(* Logix 5000 project; controller cal1632 1756-L62 rev 16.20; software revision 16.05; part 22 of 57 *)
(* tags used below, declared in another part *)
   aaa_prs : REAL;
   FAULT : BOOL;
   p01_param_fan_zero_speed : REAL;
   p01_param_open_oven_recirc_sp : REAL;
   p01_recipe_active : recipe;
   p01_sys_scp : SYS_SCP;
   p01r09_open_oven : BOOL;
   p01r09_pb_global_reset : BOOL;
   p02_dint_from_hmi : hmi_dint;
   p11r02_shutdown_temp : BOOL;
   p11r30 : routine;
   p12r02_shutdown_temp : BOOL;
   p12r30 : routine;
   p13_ai_recirc_rpm : REAL;
   p13_ao_recirc_selected_speed : REAL;
   p13_di_recirc : acs800_di_normal;
   p13_di_recirc_fan_mtr_ts : BOOL;
   p13_di_recirc_flow_ok : BOOL;
   p13_dint_to_hmi : DINT[16];
   p13_do_recirc : acs800_do_normal;
   p13r02_shutdown_temp : BOOL;
   p13r20_state : DINT;
   p13r32 : routine;
   p13r32_pb_start : BOOL;
   p13r32_pb_stop : BOOL;
   p13r32_request_auto_run : BOOL;
   p13r32_run_permissive : BOOL;
   p13r32_timer_fault : TIMER[5];
   p13r32_timer_warning : TIMER[5];
   p13r32_vfd_stopped : BOOL;
   p19_ai_prs : REAL;
   p19_ai_tc01 : REAL;
   p19_ao_cv : REAL;
   p19_di_pump : BOOL;
   p19_di_tc01_bo : BOOL;
   p19_di_tc02_bo : BOOL;
   p19_dint_to_hmi : DINT[16];
   p19_do_pump : BOOL;
   p19_flow_input_max : REAL;
   p19_flow_input_min : REAL;
   p19_flow_output_max : REAL;
   p19_flow_output_min : REAL;
   p19_param_prs_offset : REAL;
   p19_param_tc01z : REAL;
   p19_prs_input_max : REAL;
   p19_prs_input_min : REAL;
   p19_prs_output_max : REAL;
   p19_prs_output_min : REAL;
   p19r01 : routine;
   p19r02 : routine;
   p19r02_fault_exists : BOOL;
   p19r02_timer_fault : TIMER[4];
   p19r02_timer_warning : TIMER[4];
   p19r02_unack_fault : BOOL;
   p19r02_unack_warning : BOOL;
   p19r02_warning_exists : BOOL;
   p19r03 : routine;
   p19r03_flow_scp : SYS_SCP;
   p19r03_prs_input_max : REAL;
   p19r03_prs_input_min : REAL;
   p19r03_prs_output_max : REAL;
   p19r03_prs_output_min : REAL;
   p19r03_prs_scp : SYS_SCP;
   p19r03_timer_fault : TIMER[4];
   p19r03_timer_warning : TIMER[4];
   p19r04 : routine;
   p19r04_timer_fault : TIMER[4];
   p19r04_timer_warning : TIMER[4];
   p19r05 : routine;
   p19r06 : routine;
   p19r07 : routine;
   p19r08 : routine;
   p19r09 : routine;
   p19r10 : routine;
   p19r30 : routine;
   p19r31 : routine;
   p23r02 : routine;
(* P13_Zone_3, continued *)

ROUTINE R32_Recirc_VFD   (* ladder *)
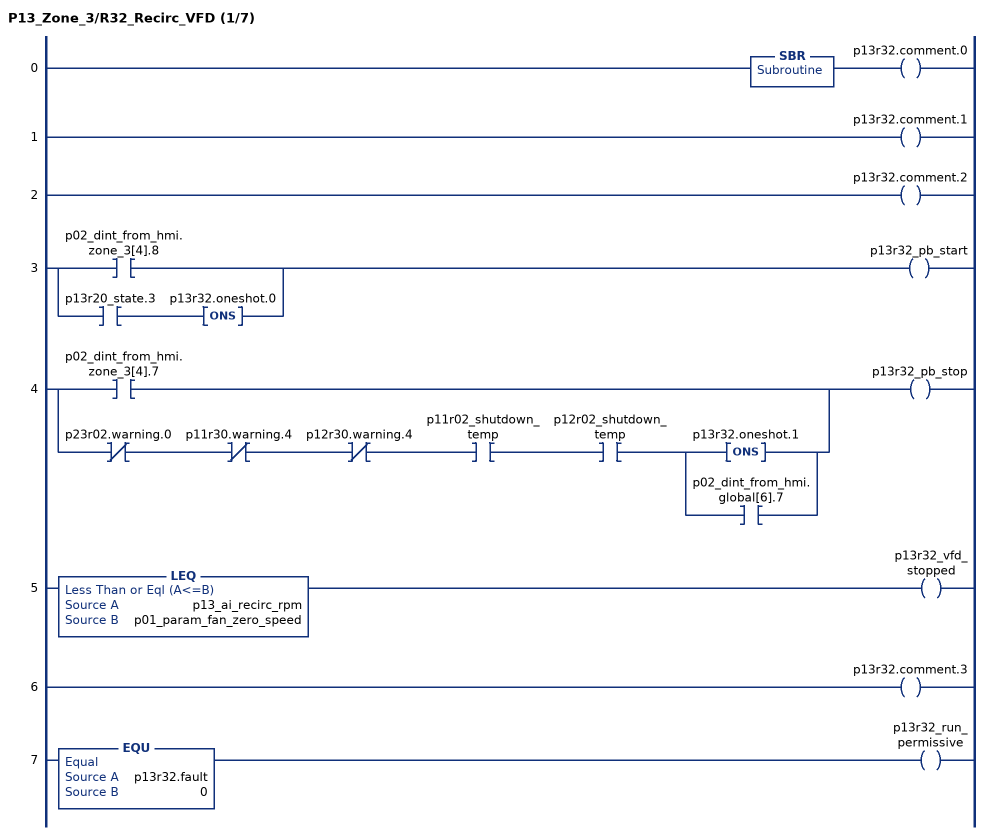
   0: SBR()OTE(p13r32.comment.0);
   1: OTE(p13r32.comment.1);
   2: OTE(p13r32.comment.2);
   3: [XIC(p02_dint_from_hmi.zone_3[4].8) ,XIC(p13r20_state.3) ONS(p13r32.oneshot.0) ]OTE(p13r32_pb_start);
   4: [XIC(p02_dint_from_hmi.zone_3[4].7) ,XIO(p23r02.warning.0) XIO(p11r30.warning.4) XIO(p12r30.warning.4) XIC(p11r02_shutdown_temp) XIC(p12r02_shutdown_temp) [ONS(p13r32.oneshot.1) ,XIC(p02_dint_from_hmi.global[6].7) ] ]OTE(p13r32_pb_stop);
   5: LEQ(p13_ai_recirc_rpm,p01_param_fan_zero_speed)OTE(p13r32_vfd_stopped);
   6: OTE(p13r32.comment.3);
   7: EQU(p13r32.fault,0)OTE(p13r32_run_permissive);
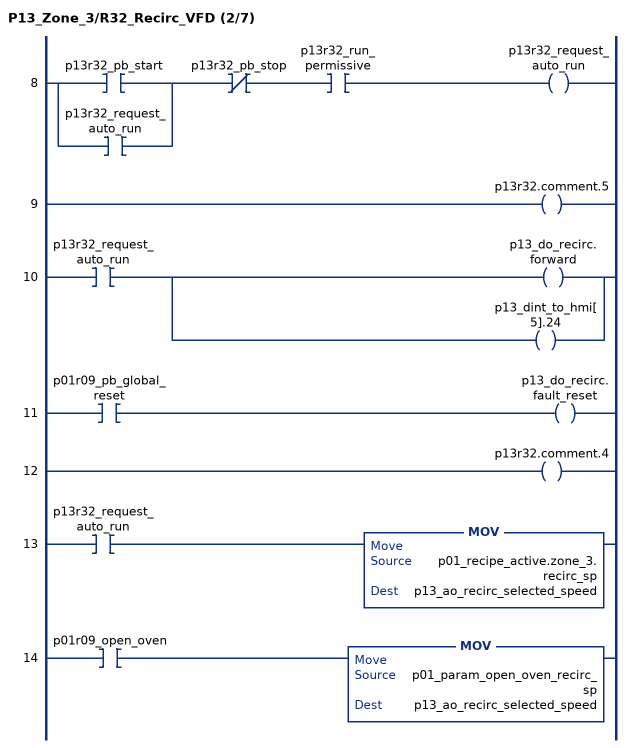
   8: [XIC(p13r32_pb_start) ,XIC(p13r32_request_auto_run) ]XIO(p13r32_pb_stop)XIC(p13r32_run_permissive)OTE(p13r32_request_auto_run);
   9: OTE(p13r32.comment.5);
   10: XIC(p13r32_request_auto_run)[OTE(p13_do_recirc.forward) ,OTE(p13_dint_to_hmi[5].24) ];
   11: XIC(p01r09_pb_global_reset)OTE(p13_do_recirc.fault_reset);
   12: OTE(p13r32.comment.4);
   13: XIC(p13r32_request_auto_run)MOV(p01_recipe_active.zone_3.recirc_sp,p13_ao_recirc_selected_speed);
   14: XIC(p01r09_open_oven)MOV(p01_param_open_oven_recirc_sp,p13_ao_recirc_selected_speed);
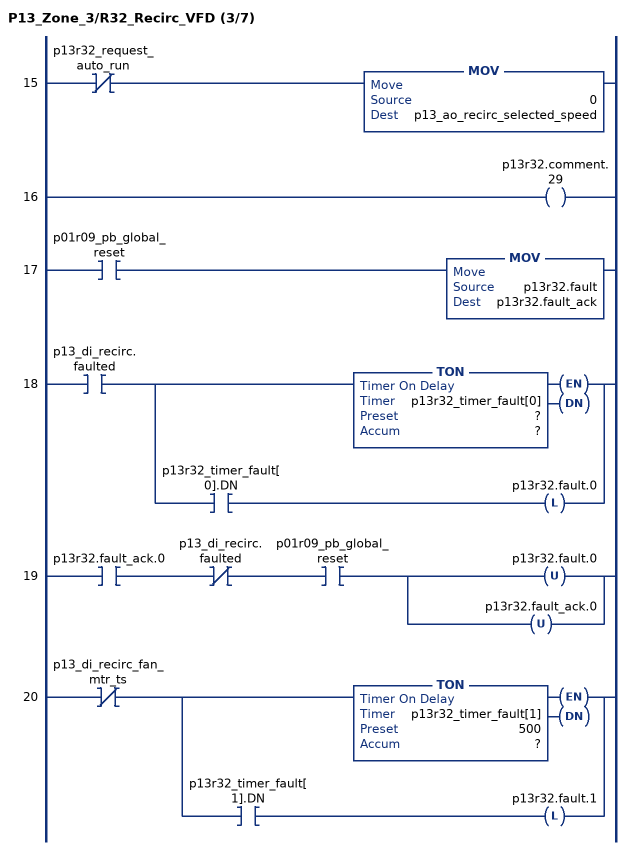
   15: XIO(p13r32_request_auto_run)MOV(0,p13_ao_recirc_selected_speed);
   16: OTE(p13r32.comment.29);
   17: XIC(p01r09_pb_global_reset)MOV(p13r32.fault,p13r32.fault_ack);
   18: XIC(p13_di_recirc.faulted)[TON(p13r32_timer_fault[0],?,?) ,XIC(p13r32_timer_fault[0].DN) OTL(p13r32.fault.0) ];
   19: XIC(p13r32.fault_ack.0)XIO(p13_di_recirc.faulted)XIC(p01r09_pb_global_reset)[OTU(p13r32.fault.0) ,OTU(p13r32.fault_ack.0) ];
   20: XIO(p13_di_recirc_fan_mtr_ts)[TON(p13r32_timer_fault[1],?,?) ,XIC(p13r32_timer_fault[1].DN) OTL(p13r32.fault.1) ];
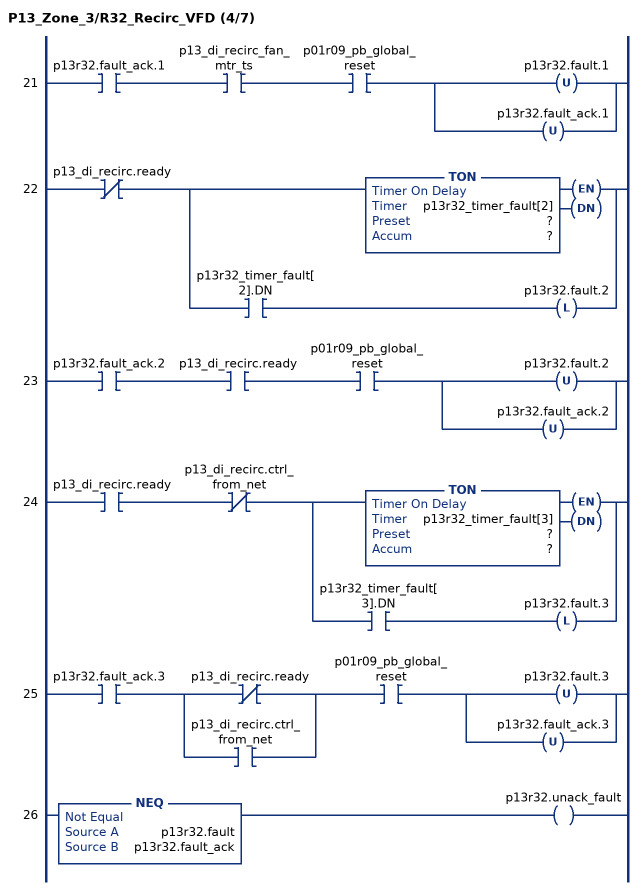
   21: XIC(p13r32.fault_ack.1)XIC(p13_di_recirc_fan_mtr_ts)XIC(p01r09_pb_global_reset)[OTU(p13r32.fault.1) ,OTU(p13r32.fault_ack.1) ];
   22: XIO(p13_di_recirc.ready)[TON(p13r32_timer_fault[2],?,?) ,XIC(p13r32_timer_fault[2].DN) OTL(p13r32.fault.2) ];
   23: XIC(p13r32.fault_ack.2)XIC(p13_di_recirc.ready)XIC(p01r09_pb_global_reset)[OTU(p13r32.fault.2) ,OTU(p13r32.fault_ack.2) ];
   24: XIC(p13_di_recirc.ready)XIO(p13_di_recirc.ctrl_from_net)[TON(p13r32_timer_fault[3],?,?) ,XIC(p13r32_timer_fault[3].DN) OTL(p13r32.fault.3) ];
   25: XIC(p13r32.fault_ack.3)[XIO(p13_di_recirc.ready) ,XIC(p13_di_recirc.ctrl_from_net) ]XIC(p01r09_pb_global_reset)[OTU(p13r32.fault.3) ,OTU(p13r32.fault_ack.3) ];
   26: NEQ(p13r32.fault,p13r32.fault_ack)OTE(p13r32.unack_fault);
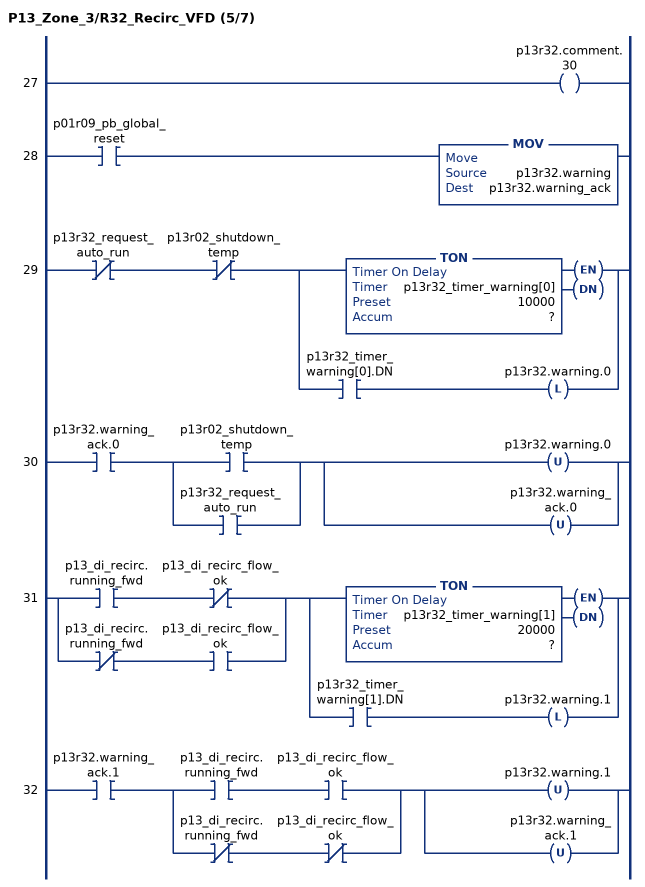
   27: OTE(p13r32.comment.30);
   28: XIC(p01r09_pb_global_reset)MOV(p13r32.warning,p13r32.warning_ack);
   29: XIO(p13r32_request_auto_run)XIO(p13r02_shutdown_temp)[TON(p13r32_timer_warning[0],?,?) ,XIC(p13r32_timer_warning[0].DN) OTL(p13r32.warning.0) ];
   30: XIC(p13r32.warning_ack.0)[XIC(p13r02_shutdown_temp) ,XIC(p13r32_request_auto_run) ][OTU(p13r32.warning.0) ,OTU(p13r32.warning_ack.0) ];
   31: [XIC(p13_di_recirc.running_fwd) XIO(p13_di_recirc_flow_ok) ,XIO(p13_di_recirc.running_fwd) XIC(p13_di_recirc_flow_ok) ][TON(p13r32_timer_warning[1],?,?) ,XIC(p13r32_timer_warning[1].DN) OTL(p13r32.warning.1) ];
   32: XIC(p13r32.warning_ack.1)[XIC(p13_di_recirc.running_fwd) XIC(p13_di_recirc_flow_ok) ,XIO(p13_di_recirc.running_fwd) XIO(p13_di_recirc_flow_ok) ][OTU(p13r32.warning.1) ,OTU(p13r32.warning_ack.1) ];
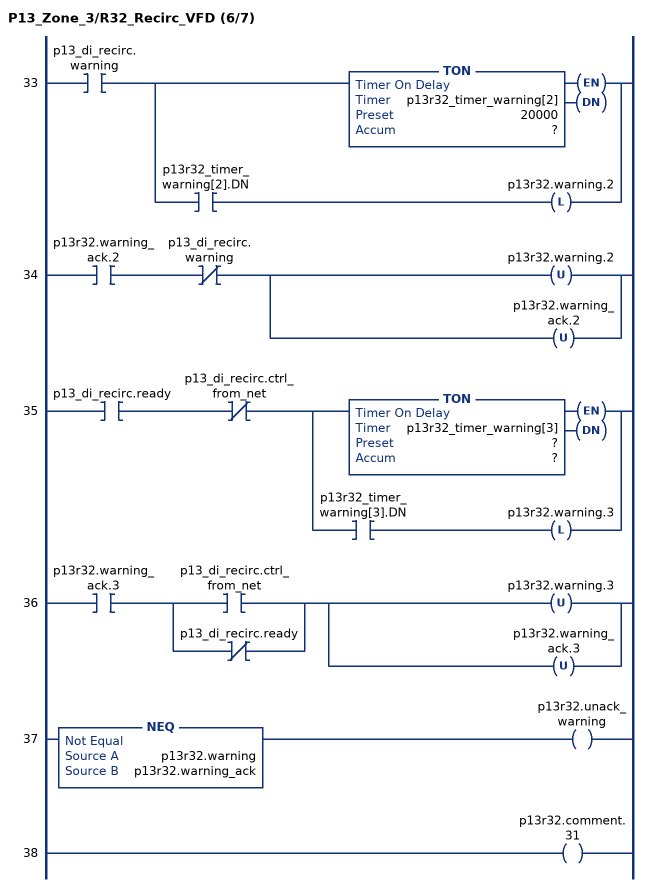
   33: XIC(p13_di_recirc.warning)[TON(p13r32_timer_warning[2],?,?) ,XIC(p13r32_timer_warning[2].DN) OTL(p13r32.warning.2) ];
   34: XIC(p13r32.warning_ack.2)XIO(p13_di_recirc.warning)[OTU(p13r32.warning.2) ,OTU(p13r32.warning_ack.2) ];
   35: XIC(p13_di_recirc.ready)XIO(p13_di_recirc.ctrl_from_net)[TON(p13r32_timer_warning[3],?,?) ,XIC(p13r32_timer_warning[3].DN) OTL(p13r32.warning.3) ];
   36: XIC(p13r32.warning_ack.3)[XIC(p13_di_recirc.ctrl_from_net) ,XIO(p13_di_recirc.ready) ][OTU(p13r32.warning.3) ,OTU(p13r32.warning_ack.3) ];
   37: NEQ(p13r32.warning,p13r32.warning_ack)OTE(p13r32.unack_warning);
   38: OTE(p13r32.comment.31);
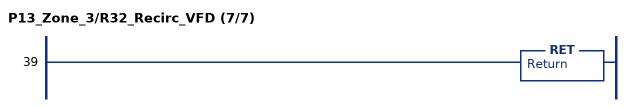
   39: RET();
END_ROUTINE
END_PROGRAM

PROGRAM P19_Advanced_Cooling   (* main routine R01_Main *)

ROUTINE R01_Main   (* ladder *)
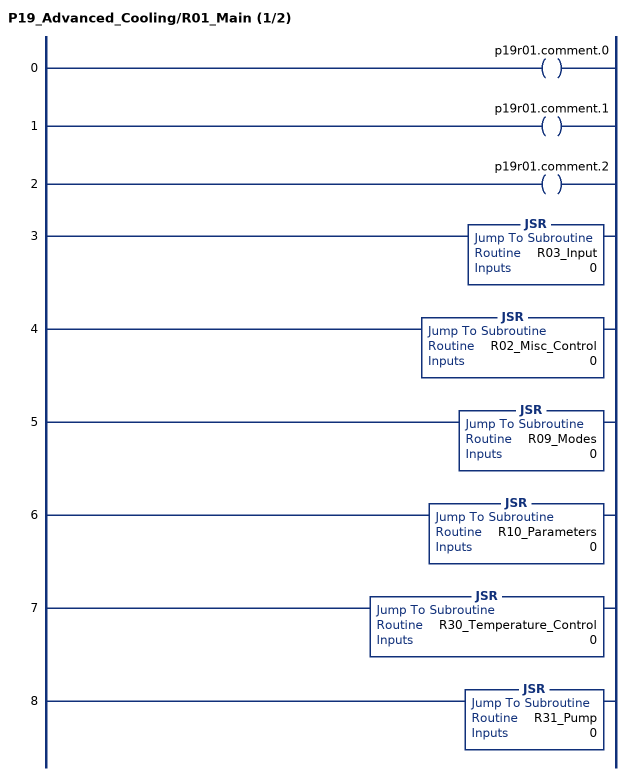
   0: OTE(p19r01.comment.0);
   1: OTE(p19r01.comment.1);
   2: OTE(p19r01.comment.2);
   3: JSR(R03_Input,0);
   4: JSR(R02_Misc_Control,0);
   5: JSR(R09_Modes,0);
   6: JSR(R10_Parameters,0);
   7: JSR(R30_Temperature_Control,0);
   8: JSR(R31_Pump,0);
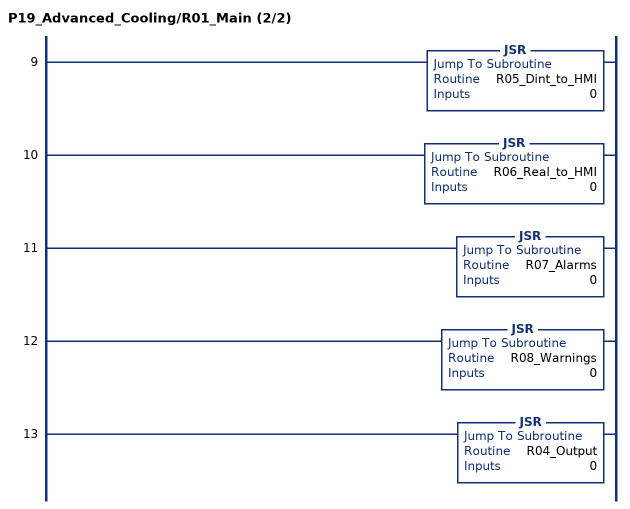
   9: JSR(R05_Dint_to_HMI,0);
   10: JSR(R06_Real_to_HMI,0);
   11: JSR(R07_Alarms,0);
   12: JSR(R08_Warnings,0);
   13: JSR(R04_Output,0);
END_ROUTINE

ROUTINE R02_Misc_Control   (* ladder *)
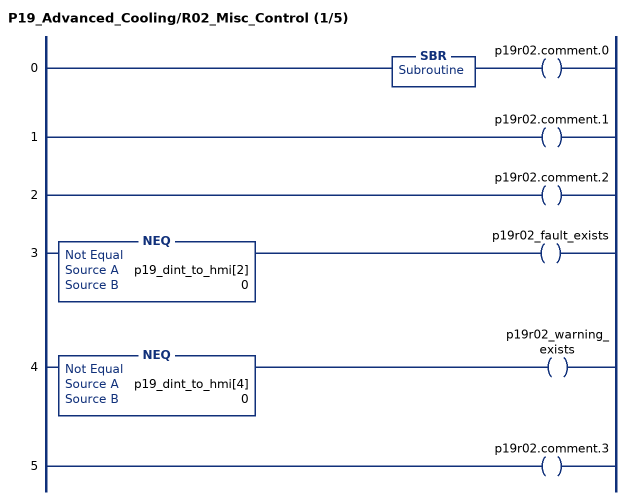
   0: SBR()OTE(p19r02.comment.0);
   1: OTE(p19r02.comment.1);
   2: OTE(p19r02.comment.2);
   3: NEQ(p19_dint_to_hmi[2],0)OTE(p19r02_fault_exists);
   4: NEQ(p19_dint_to_hmi[4],0)OTE(p19r02_warning_exists);
   5: OTE(p19r02.comment.3);
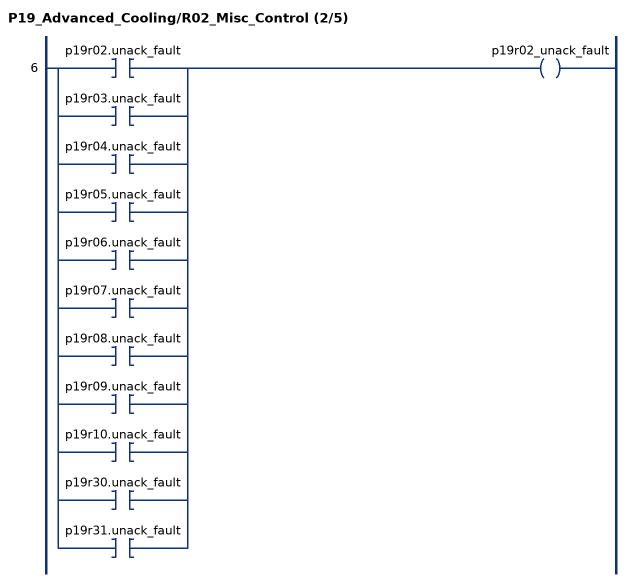
   6: [XIC(p19r02.unack_fault) ,XIC(p19r03.unack_fault) ,XIC(p19r04.unack_fault) ,XIC(p19r05.unack_fault) ,XIC(p19r06.unack_fault) ,XIC(p19r07.unack_fault) ,XIC(p19r08.unack_fault) ,XIC(p19r09.unack_fault) ,XIC(p19r10.unack_fault) ,XIC(p19r30.unack_fault) ,XIC(p19r31.unack_fault) ]OTE(p19r02_unack_fault);
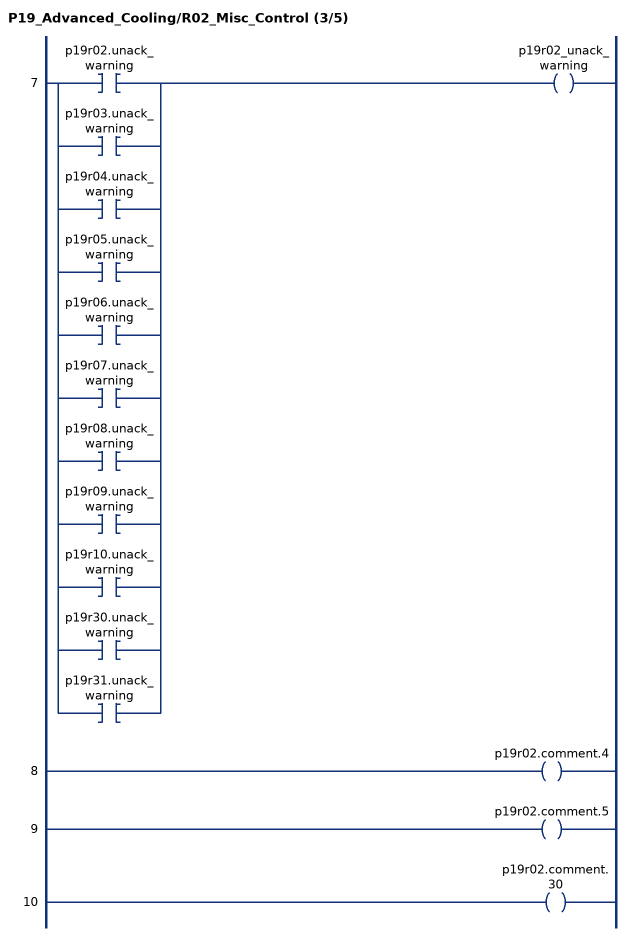
   7: [XIC(p19r02.unack_warning) ,XIC(p19r03.unack_warning) ,XIC(p19r04.unack_warning) ,XIC(p19r05.unack_warning) ,XIC(p19r06.unack_warning) ,XIC(p19r07.unack_warning) ,XIC(p19r08.unack_warning) ,XIC(p19r09.unack_warning) ,XIC(p19r10.unack_warning) ,XIC(p19r30.unack_warning) ,XIC(p19r31.unack_warning) ]OTE(p19r02_unack_warning);
   8: OTE(p19r02.comment.4);
   9: OTE(p19r02.comment.5);
   10: OTE(p19r02.comment.30);
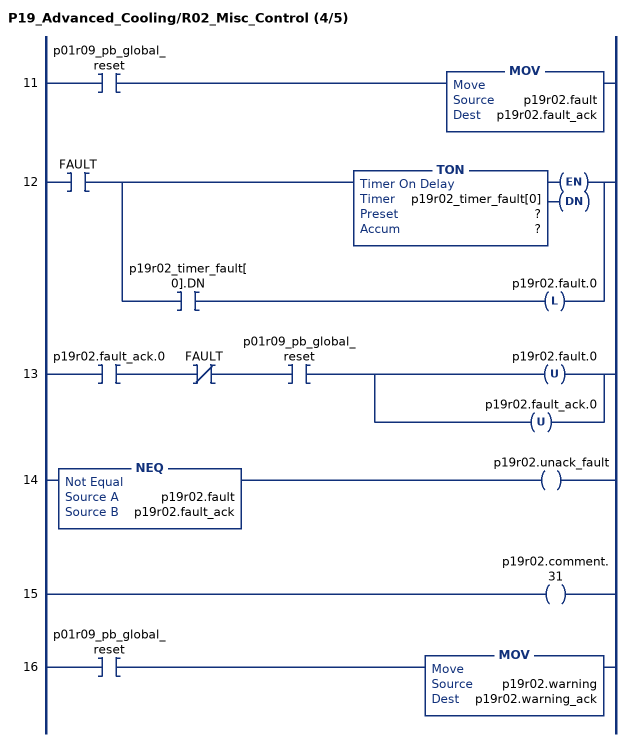
   11: XIC(p01r09_pb_global_reset)MOV(p19r02.fault,p19r02.fault_ack);
   12: XIC(FAULT)[TON(p19r02_timer_fault[0],?,?) ,XIC(p19r02_timer_fault[0].DN) OTL(p19r02.fault.0) ];
   13: XIC(p19r02.fault_ack.0)XIO(FAULT)XIC(p01r09_pb_global_reset)[OTU(p19r02.fault.0) ,OTU(p19r02.fault_ack.0) ];
   14: NEQ(p19r02.fault,p19r02.fault_ack)OTE(p19r02.unack_fault);
   15: OTE(p19r02.comment.31);
   16: XIC(p01r09_pb_global_reset)MOV(p19r02.warning,p19r02.warning_ack);
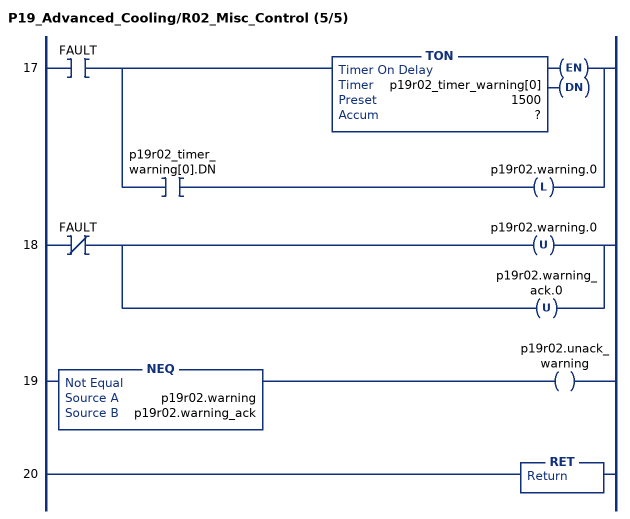
   17: XIC(FAULT)[TON(p19r02_timer_warning[0],?,?) ,XIC(p19r02_timer_warning[0].DN) OTL(p19r02.warning.0) ];
   18: XIO(FAULT)[OTU(p19r02.warning.0) ,OTU(p19r02.warning_ack.0) ];
   19: NEQ(p19r02.warning,p19r02.warning_ack)OTE(p19r02.unack_warning);
   20: RET();
END_ROUTINE

ROUTINE R03_Input   (* ladder *)
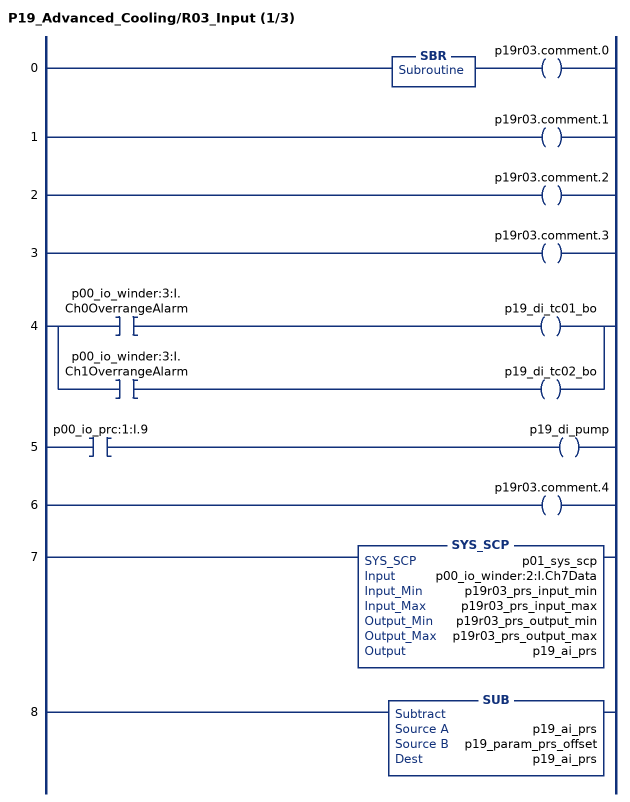
   0: SBR()OTE(p19r03.comment.0);
   1: OTE(p19r03.comment.1);
   2: OTE(p19r03.comment.2);
   3: OTE(p19r03.comment.3);
   4: [XIC(p00_io_winder:3:I.Ch0OverrangeAlarm) OTE(p19_di_tc01_bo) ,XIC(p00_io_winder:3:I.Ch1OverrangeAlarm) OTE(p19_di_tc02_bo) ];
   5: XIC(p00_io_prc:1:I.9)OTE(p19_di_pump);
   6: OTE(p19r03.comment.4);
   7: SYS_SCP(p01_sys_scp,p00_io_winder:2:I.Ch7Data,p19r03_prs_input_min,p19r03_prs_input_max,p19r03_prs_output_min,p19r03_prs_output_max,p19_ai_prs);
   8: SUB(p19_ai_prs,p19_param_prs_offset,p19_ai_prs);
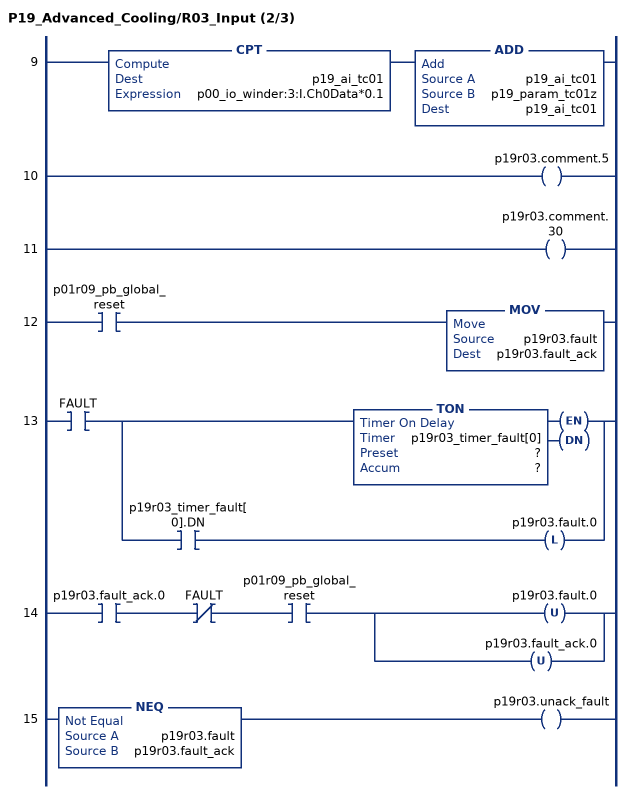
   9: CPT(p19_ai_tc01,p00_io_winder:3:I.Ch0Data*0.1)ADD(p19_ai_tc01,p19_param_tc01z,p19_ai_tc01);
   10: OTE(p19r03.comment.5);
   11: OTE(p19r03.comment.30);
   12: XIC(p01r09_pb_global_reset)MOV(p19r03.fault,p19r03.fault_ack);
   13: XIC(FAULT)[TON(p19r03_timer_fault[0],?,?) ,XIC(p19r03_timer_fault[0].DN) OTL(p19r03.fault.0) ];
   14: XIC(p19r03.fault_ack.0)XIO(FAULT)XIC(p01r09_pb_global_reset)[OTU(p19r03.fault.0) ,OTU(p19r03.fault_ack.0) ];
   15: NEQ(p19r03.fault,p19r03.fault_ack)OTE(p19r03.unack_fault);
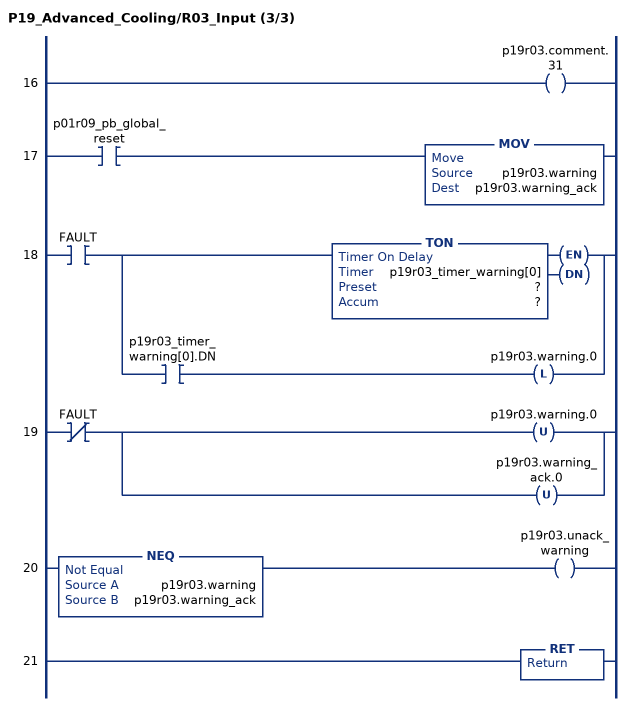
   16: OTE(p19r03.comment.31);
   17: XIC(p01r09_pb_global_reset)MOV(p19r03.warning,p19r03.warning_ack);
   18: XIC(FAULT)[TON(p19r03_timer_warning[0],?,?) ,XIC(p19r03_timer_warning[0].DN) OTL(p19r03.warning.0) ];
   19: XIO(FAULT)[OTU(p19r03.warning.0) ,OTU(p19r03.warning_ack.0) ];
   20: NEQ(p19r03.warning,p19r03.warning_ack)OTE(p19r03.unack_warning);
   21: RET();
END_ROUTINE

ROUTINE R04_Output   (* ladder *)
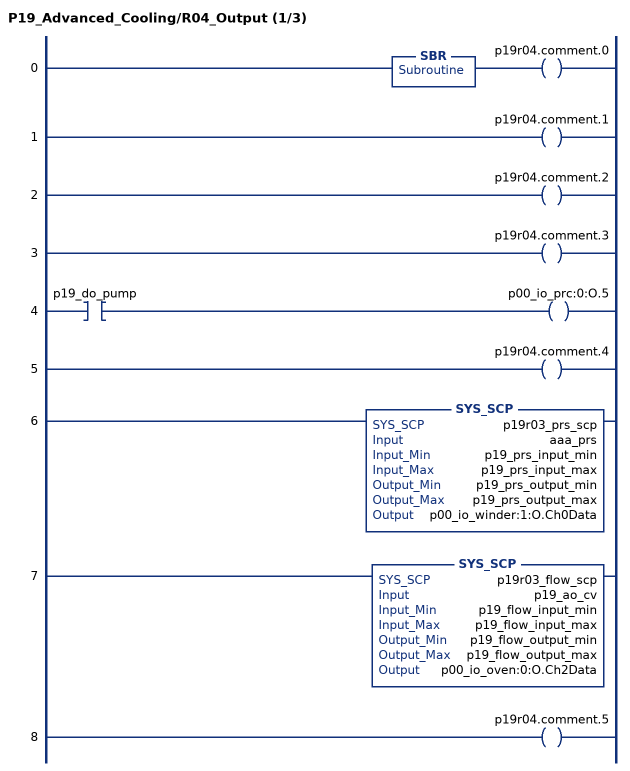
   0: SBR()OTE(p19r04.comment.0);
   1: OTE(p19r04.comment.1);
   2: OTE(p19r04.comment.2);
   3: OTE(p19r04.comment.3);
   4: XIC(p19_do_pump)OTE(p00_io_prc:0:O.5);
   5: OTE(p19r04.comment.4);
   6: SYS_SCP(p19r03_prs_scp,aaa_prs,p19_prs_input_min,p19_prs_input_max,p19_prs_output_min,p19_prs_output_max,p00_io_winder:1:O.Ch0Data);
   7: SYS_SCP(p19r03_flow_scp,p19_ao_cv,p19_flow_input_min,p19_flow_input_max,p19_flow_output_min,p19_flow_output_max,p00_io_oven:0:O.Ch2Data);
   8: OTE(p19r04.comment.5);
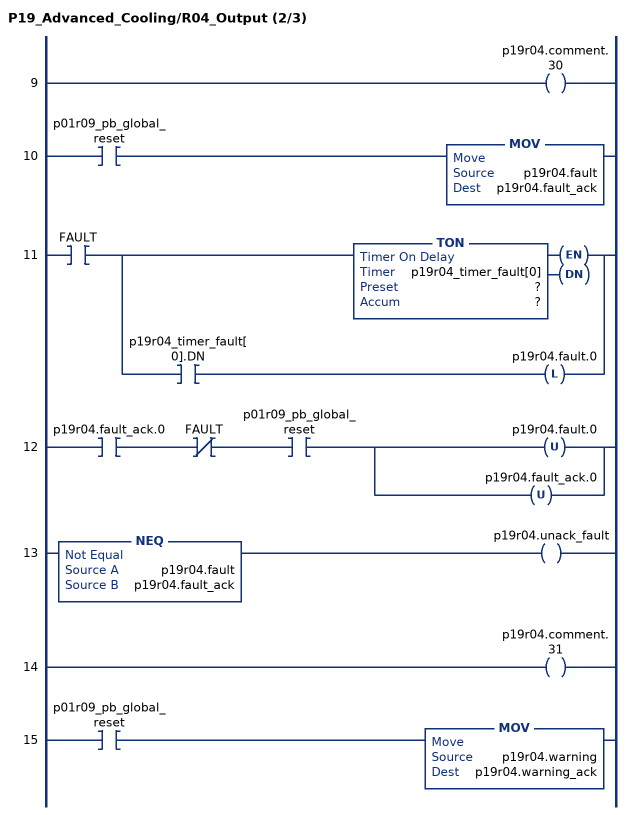
   9: OTE(p19r04.comment.30);
   10: XIC(p01r09_pb_global_reset)MOV(p19r04.fault,p19r04.fault_ack);
   11: XIC(FAULT)[TON(p19r04_timer_fault[0],?,?) ,XIC(p19r04_timer_fault[0].DN) OTL(p19r04.fault.0) ];
   12: XIC(p19r04.fault_ack.0)XIO(FAULT)XIC(p01r09_pb_global_reset)[OTU(p19r04.fault.0) ,OTU(p19r04.fault_ack.0) ];
   13: NEQ(p19r04.fault,p19r04.fault_ack)OTE(p19r04.unack_fault);
   14: OTE(p19r04.comment.31);
   15: XIC(p01r09_pb_global_reset)MOV(p19r04.warning,p19r04.warning_ack);
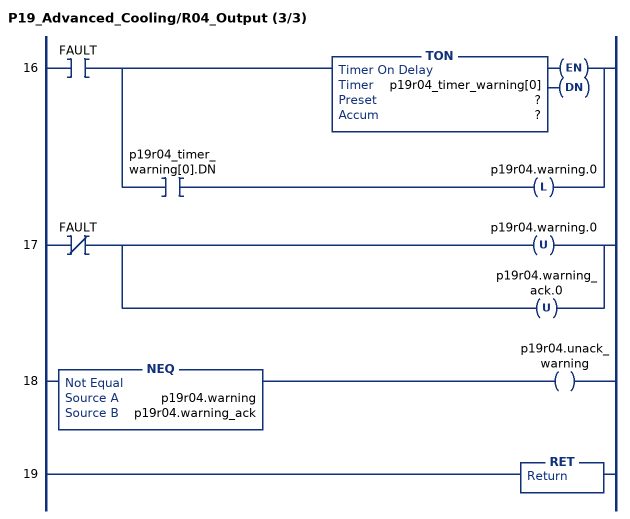
   16: XIC(FAULT)[TON(p19r04_timer_warning[0],?,?) ,XIC(p19r04_timer_warning[0].DN) OTL(p19r04.warning.0) ];
   17: XIO(FAULT)[OTU(p19r04.warning.0) ,OTU(p19r04.warning_ack.0) ];
   18: NEQ(p19r04.warning,p19r04.warning_ack)OTE(p19r04.unack_warning);
   19: RET();
END_ROUTINE
